FUNCTION F_ContinousResultID : bool
VAR_INPUT
	nCurrentResultID :UINT;
	nPreviousResultID: UINT;
	END_VAR
VAR
	bIsContinuous : BOOL; 

END_VAR

IF nPreviousResultID = 32767 THEN
    // Ha az előző ID 32767, akkor a következőnek 0-nak kell lennie
    bIsContinuous := (nCurrentResultID = 0);
ELSE
    // Általános eset: az aktuális ID az előző + 1 legyen
    bIsContinuous := (nCurrentResultID = nPreviousResultID + 1);
END_IF

F_ContinousResultID:= bIsContinuous;

END_FUNCTION

(* stored: Version 1.1.0.1, ProductVersion 3.1.4024.14
   POU F_ContinousResultID: Id {e84588e8-e050-4cd8-a74f-8b3ee022c90c}, SpecialFunc None *)
